TYPE ZCom :
STRUCT
  // module context
  App : ZApplication.ApplicationComPublish;
  Alarming : ZApplication.AlarmingCom;
  Messages : ZApplication.MessagingCom;
  
  // unit context
  Unit : ZComUnit;

END_STRUCT
END_TYPE

(* stored: Version 1.1.0.1
   DUT ZCom: Id {3290ec21-ae73-4dc7-b3a8-0907d1ae3a7b} *)
